# EPICS autosave request: mw100App/Db/MW100_DAC_slot2_settings.req
$(P)$(DAU):011:Label
$(P)$(DAU):012:Label
$(P)$(DAU):013:Label
$(P)$(DAU):014:Label
$(P)$(DAU):015:Label
$(P)$(DAU):016:Label
$(P)$(DAU):017:Label
$(P)$(DAU):018:Label
